{attribute 'qualified_only'}
{attribute 'to_string'}
TYPE E_AxisNames :
(
	None := 0,
	IncSlits_X_Translation := 1,
	IncSlits_Z_Translation :=2,
	IncSlits_North := 3,
	IncSlits_South := 4,
	IncSlits_East := 5,
	IncSlits_West := 6,
	Sample_Stack_X_Translation := 7,
	Sample_Stack_Y_Translation := 8,
	Tomography_Phi := 9,
	Tomography_Chi := 10,
	Tomography_Theta := 11,
	SampleEnv_ExtraAxes := 12,
	Camera_LensAdj := 13,
	Camera_FlipRot := 14, // check correct
	Camera_Tilt := 15, //check correct
	Sample_Stack_Z_Translation :=16,
	Sample_Stack_Z_Rotation :=17,
	Coll_North_X :=18,
	Coll_North_Y :=19,
	Coll_South_X :=20,
	Coll_South_Y :=21,
	PinholeSelector := 22,
	Monitor5 := 23,
	Slit_1_North := 24,
	Slit_1_South := 25,
	Slit_1_East := 26,
	Slit_1_West := 27,
	Slit_2_North := 28,
	Slit_2_South := 29,
	Slit_2_East := 30,
	Slit_2_West := 31,
	Slit_3_North := 32,
	Slit_3_South := 33,
	Slit_3_East := 34,
	Slit_3_West := 35,
	Slit_4_North := 36,
	Slit_4_South := 37,
	Slit_4_East := 38,
	Slit_4_West := 39,
	Slit_5_North := 40,
	Slit_5_South := 41,
	Slit_5_East := 42,
	Slit_5_West := 43
);
END_TYPE

(* stored: Version 1.1.0.1, ProductVersion 3.1.4026.18
   DUT E_AxisNames: Id {51d6d500-1f76-496d-ac31-56a31f33e006} *)
